KUKA KRL data list: EKITEST.DAT

&ACCESS RVP
&REL 1
DEFDAT EKITEST
ENDDAT
